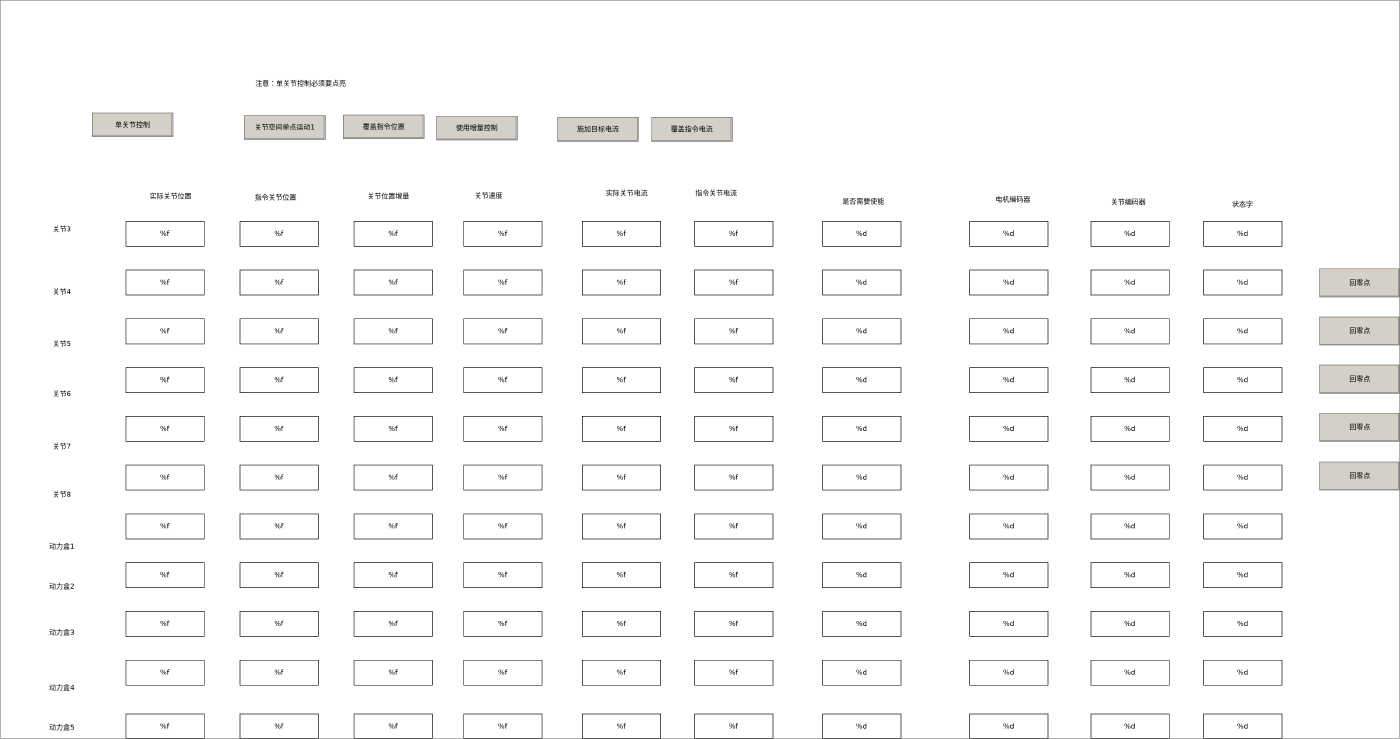
VISUALIZATION motion_a2  // 2208x1167
    Button (385,182 128x38), "关节空间单点运动1", colour toggle: g_motionTest.m_uiArmMode[2,1]
        tap g_motionTest.m_uiArmMode[1,1]
    Label (362,298 145x28), "指令关节位置"
    Label (194,295 150x30), "实际关节位置"
    Label (540,296 145x28), "关节位置增量"
    Label (698,295 145x28), "关节速度"
    Label (916,291 145x28), "实际关节电流"
    Label (1057,291 145x28), "指令关节电流"
    Rectangle (198,580 124x40), "%f", text variable: g_motionTest.m_actJntPos[2][1]
    Label (25,348 145x28), "关节3"
    Label (25,447 145x28), "关节4"
    Label (25,529 145x28), "关节5"
    Label (25,608 145x28), "关节6"
    Label (25,691 145x28), "关节7"
    Label (25,767 145x28), "关节8"
    Label (25,849 145x28), "动力盒1"
    Label (25,912 145x28), "动力盒2"
    Label (25,1135 145x28), "动力盒5"
    Label (25,985 145x28), "动力盒3"
    Label (25,1072 145x28), "动力盒4"
    Rectangle (198,657 124x40), "%f", text variable: g_motionTest.m_actJntPos[2][2]
    Rectangle (198,734 124x40), "%f", text variable: g_motionTest.m_actJntPos[2][3]
    Rectangle (198,811 124x40), "%f", text variable: g_motionTest.m_actJntPos[2][4]
    Rectangle (198,888 124x40), "%f", text variable: g_motionTest.m_actJntPos[2][5]
    Rectangle (198,965 124x40), "%f", text variable: g_motionTest.m_actJntPos[2][6]
    Rectangle (198,1042 124x40), "%f", text variable: g_motionTest.m_actJntPos[2][7]
    Rectangle (198,1127 124x40), "%f", text variable: g_motionTest.m_actJntPos[2][8]
    Rectangle (198,349 124x40), "%f", text variable: g_motionTest.m_actJntPosSetup[2][3]
    Rectangle (198,426 124x40), "%f", text variable: g_motionTest.m_actJntPosSetup[2][4]
    Rectangle (198,503 124x40), "%f", text variable: g_motionTest.m_actJntPosSetup[2][5]
    Rectangle (378,349 124x40), "%f", text variable: g_motionTest.m_targetJntPosSetup[2][3]
        OnMouseClick: write the text variable via Default
    Rectangle (378,426 124x40), "%f", text variable: g_motionTest.m_targetJntPosSetup[2][4]
        OnMouseClick: write the text variable via Default
    Rectangle (378,503 124x40), "%f", text variable: g_motionTest.m_targetJntPosSetup[2][5]
        OnMouseClick: write the text variable via Default
    Rectangle (378,580 124x40), "%f", text variable: g_motionTest.m_targetJntPosN8[2][1]
        OnMouseClick: write the text variable via Default
    Rectangle (378,657 124x40), "%f", text variable: g_motionTest.m_targetJntPosN8[2][2]
        OnMouseClick: write the text variable via Default
    Rectangle (378,734 124x40), "%f", text variable: g_motionTest.m_targetJntPosN8[2][3]
        OnMouseClick: write the text variable via Default
    Rectangle (378,811 124x40), "%f", text variable: g_motionTest.m_targetJntPosN8[2][4]
        OnMouseClick: write the text variable via Default
    Rectangle (378,888 124x40), "%f", text variable: g_motionTest.m_targetJntPosN8[2][5]
        OnMouseClick: write the text variable via Default
    Rectangle (378,965 124x40), "%f", text variable: g_motionTest.m_targetJntPosN8[2][6]
        OnMouseClick: write the text variable via Default
    Rectangle (378,1042 124x40), "%f", text variable: g_motionTest.m_targetJntPosN8[2][7]
        OnMouseClick: write the text variable via Default
    Rectangle (378,1127 124x40), "%f", text variable: g_motionTest.m_targetJntPosN8[2][8]
        OnMouseClick: write the text variable via Default
    Rectangle (558,349 124x40), "%f", text variable: g_motionTest.m_targetJntPosIncSetup[2][3]
        OnMouseClick: write the text variable via Default
    Rectangle (558,426 124x40), "%f", text variable: g_motionTest.m_targetJntPosIncSetup[2][4]
        OnMouseClick: write the text variable via Default
    Rectangle (558,503 124x40), "%f", text variable: g_motionTest.m_targetJntPosIncSetup[2][5]
        OnMouseClick: write the text variable via Default
    Rectangle (558,580 124x40), "%f", text variable: g_motionTest.m_targetJntPosIncN8[2][1]
        OnMouseClick: write the text variable via Default
    Rectangle (558,657 124x40), "%f", text variable: g_motionTest.m_targetJntPosIncN8[2][2]
        OnMouseClick: write the text variable via Default
    Rectangle (558,734 124x40), "%f", text variable: g_motionTest.m_targetJntPosIncN8[2][3]
        OnMouseClick: write the text variable via Default
    Rectangle (558,811 124x40), "%f", text variable: g_motionTest.m_targetJntPosIncN8[2][4]
        OnMouseClick: write the text variable via Default
    Rectangle (558,888 124x40), "%f", text variable: g_motionTest.m_targetJntPosIncN8[2][5]
        OnMouseClick: write the text variable via Default
    Rectangle (558,965 124x40), "%f", text variable: g_motionTest.m_targetJntPosIncN8[2][6]
        OnMouseClick: write the text variable via Default
    Rectangle (558,1042 124x40), "%f", text variable: g_motionTest.m_targetJntPosIncN8[2][7]
        OnMouseClick: write the text variable via Default
    Rectangle (558,1127 124x40), "%f", text variable: g_motionTest.m_targetJntPosIncN8[2][8]
        OnMouseClick: write the text variable via Default
    Rectangle (731,349 124x40), "%f", text variable: g_motionTest.m_targetJntVelSetup[2][3]
        OnMouseClick: write the text variable via Default
    Rectangle (731,426 124x40), "%f", text variable: g_motionTest.m_targetJntVelSetup[2][4]
        OnMouseClick: write the text variable via Default
    Rectangle (731,503 124x40), "%f", text variable: g_motionTest.m_targetJntVelSetup[2][5]
        OnMouseClick: write the text variable via Default
    Rectangle (731,580 124x40), "%f", text variable: g_motionTest.m_targetJntVel[2][1]
        OnMouseClick: write the text variable via Default
    Rectangle (731,657 124x40), "%f", text variable: g_motionTest.m_targetJntVel[2][2]
        OnMouseClick: write the text variable via Default
    Rectangle (731,734 124x40), "%f", text variable: g_motionTest.m_targetJntVel[2][3]
        OnMouseClick: write the text variable via Default
    Rectangle (731,811 124x40), "%f", text variable: g_motionTest.m_targetJntVel[2][4]
        OnMouseClick: write the text variable via Default
    Rectangle (731,888 124x40), "%f", text variable: g_motionTest.m_targetJntVel[2][5]
        OnMouseClick: write the text variable via Default
    Rectangle (731,965 124x40), "%f", text variable: g_motionTest.m_targetJntVel[2][6]
        OnMouseClick: write the text variable via Default
    Rectangle (731,1042 124x40), "%f", text variable: g_motionTest.m_targetJntVel[2][7]
        OnMouseClick: write the text variable via Default
    Rectangle (731,1127 124x40), "%f", text variable: g_motionTest.m_targetJntVel[2][8]
        OnMouseClick: write the text variable via Default
    Rectangle (918,349 124x40), "%f", text variable: g_motionTest.m_actJntCurrentSetup[2][3]
    Rectangle (918,426 124x40), "%f", text variable: g_motionTest.m_actJntCurrentSetup[2][4]
    Rectangle (918,503 124x40), "%f", text variable: g_motionTest.m_actJntCurrentSetup[2][5]
    Rectangle (918,580 124x40), "%f", text variable: g_motionTest.m_actJntCurrent[2][1]
    Rectangle (918,657 124x40), "%f", text variable: g_motionTest.m_actJntCurrent[2][2]
    Rectangle (918,734 124x40), "%f", text variable: g_motionTest.m_actJntCurrent[2][3]
    Rectangle (918,811 124x40), "%f", text variable: g_motionTest.m_actJntCurrent[2][4]
    Rectangle (918,888 124x40), "%f", text variable: g_motionTest.m_actJntCurrent[2][5]
    Rectangle (918,965 124x40), "%f", text variable: g_motionTest.m_actJntCurrent[2][6]
    Rectangle (918,1042 124x40), "%f", text variable: g_motionTest.m_actJntCurrent[2][7]
    Rectangle (918,1127 124x40), "%f", text variable: g_motionTest.m_actJntCurrent[2][8]
    Rectangle (1095,349 124x40), "%f", text variable: g_motionTest.m_targetJntCurrentSetup[2][3]
        OnMouseClick: write the text variable via Default
    Rectangle (1095,426 124x40), "%f", text variable: g_motionTest.m_targetJntCurrentSetup[2][4]
        OnMouseClick: write the text variable via Default
    Rectangle (1095,503 124x40), "%f", text variable: g_motionTest.m_targetJntCurrentSetup[2][5]
        OnMouseClick: write the text variable via Default
    Rectangle (1095,580 124x40), "%f", text variable: g_motionTest.m_targetJntCurrentN8[2][1]
        OnMouseClick: write the text variable via Default
    Rectangle (1095,657 124x40), "%f", text variable: g_motionTest.m_targetJntCurrentN8[2][2]
        OnMouseClick: write the text variable via Default
    Rectangle (1095,734 124x40), "%f", text variable: g_motionTest.m_targetJntCurrentN8[2][3]
        OnMouseClick: write the text variable via Default
    Rectangle (1095,811 124x40), "%f", text variable: g_motionTest.m_targetJntCurrentN8[2][4]
        OnMouseClick: write the text variable via Default
    Rectangle (1095,888 124x40), "%f", text variable: g_motionTest.m_targetJntCurrentN8[2][5]
        OnMouseClick: write the text variable via Default
    Rectangle (1095,965 124x40), "%f", text variable: g_motionTest.m_targetJntCurrentN8[2][6]
        OnMouseClick: write the text variable via Default
    Rectangle (1095,1042 124x40), "%f", text variable: g_motionTest.m_targetJntCurrentN8[2][7]
        OnMouseClick: write the text variable via Default
    Rectangle (1095,1127 124x40), "%f", text variable: g_motionTest.m_targetJntCurrentN8[2][8]
        OnMouseClick: write the text variable via Default
    Button (688,183 128x38), "使用增量控制", colour toggle: g_motionTest.m_singleMotorIncControl[2]
        toggle g_motionTest.m_singleMotorIncControl[2]
    Button (879,185 128x38), "施加目标电流", colour toggle: g_motionTest.m_uiArmMode[2,9]
        toggle g_motionTest.m_uiArmMode[2,9]
    Button (145,178 128x38), "单关节控制", colour toggle: g_motionTest.m_singleMotorControl[2]
        toggle g_motionTest.m_singleMotorControl[2]
    Label (364,117 220x30), "注意：单关节控制必须要点亮"
    Label (1289,303 145x30), "是否需要使能"
    Rectangle (1297,349 124x40), "%d", text variable: g_motionTest.m_jntEnableSetup[2][3]
        OnMouseClick: write the text variable via Default
    Rectangle (1297,426 124x40), "%d", text variable: g_motionTest.m_jntEnableSetup[2][4]
        OnMouseClick: write the text variable via Default
    Rectangle (1297,503 124x40), "%d", text variable: g_motionTest.m_jntEnableSetup[2][5]
        OnMouseClick: write the text variable via Default
    Rectangle (1297,580 124x40), "%d", text variable: g_motionTest.m_jntEnable[2][1]
        OnMouseClick: write the text variable via Default
    Rectangle (1297,657 124x40), "%d", text variable: g_motionTest.m_jntEnable[2][2]
        OnMouseClick: write the text variable via Default
    Label (1525,301 145x28), "电机编码器"
    Label (1707,305 145x28), "关节编码器"
    Label (1887,309 145x28), "状态字"
    Rectangle (1529,349 124x40), "%d", text variable: g_systemInfo.m_setupJntInfo[2,3].m_motorInput.m_motorEncoder
    Rectangle (1529,426 124x40), "%d", text variable: g_systemInfo.m_setupJntInfo[2,4].m_motorInput.m_motorEncoder
    Rectangle (1529,503 124x40), "%d", text variable: g_systemInfo.m_setupJntInfo[2,5].m_motorInput.m_motorEncoder
    Rectangle (1529,580 124x40), "%d", text variable: g_systemInfo.m_slaveJntInfo[2,1].m_motorInput.m_motorEncoder
    Rectangle (1529,657 124x40), "%d", text variable: g_systemInfo.m_slaveJntInfo[2,2].m_motorInput.m_motorEncoder
    Rectangle (1720,349 124x40), "%d", text variable: g_systemInfo.m_setupJntInfo[2,3].m_motorInput.m_linkEncoder
    Rectangle (1720,426 124x40), "%d", text variable: g_systemInfo.m_setupJntInfo[2,4].m_motorInput.m_linkEncoder
    Rectangle (1720,503 124x40), "%d", text variable: g_systemInfo.m_setupJntInfo[2,5].m_motorInput.m_linkEncoder
    Rectangle (1720,580 124x40), "%d", text variable: g_systemInfo.m_slaveJntInfo[2,1].m_motorInput.m_linkEncoder
    Rectangle (1720,657 124x40), "%d", text variable: g_systemInfo.m_slaveJntInfo[2,2].m_motorInput.m_linkEncoder
    Rectangle (1898,349 124x40), "%d", text variable: g_systemInfo.m_setupJntInfo[2,3].m_motorInput.m_statusWord
    Rectangle (1898,426 124x40), "%d", text variable: g_systemInfo.m_setupJntInfo[2,4].m_motorInput.m_statusWord
    Rectangle (1898,503 124x40), "%d", text variable: g_systemInfo.m_setupJntInfo[2,5].m_motorInput.m_statusWord
    Rectangle (1898,580 124x40), "%d", text variable: g_systemInfo.m_slaveJntInfo[2,1].m_motorInput.m_statusWord
    Rectangle (1898,657 124x40), "%d", text variable: g_systemInfo.m_slaveJntInfo[2,2].m_motorInput.m_statusWord
    Rectangle (1529,734 124x40), "%d", text variable: g_systemInfo.m_slaveJntInfo[2,3].m_motorInput.m_motorEncoder
    Rectangle (1529,811 124x40), "%d", text variable: g_systemInfo.m_slaveJntInfo[2,4].m_motorInput.m_motorEncoder
    Rectangle (1529,888 124x40), "%d", text variable: g_systemInfo.m_slaveJntInfo[2,5].m_motorInput.m_motorEncoder
    Rectangle (1529,965 124x40), "%d", text variable: g_systemInfo.m_slaveJntInfo[2,6].m_motorInput.m_motorEncoder
    Rectangle (1529,1042 124x40), "%d", text variable: g_systemInfo.m_slaveJntInfo[2,7].m_motorInput.m_motorEncoder
    Rectangle (1529,1127 124x40), "%d", text variable: g_systemInfo.m_slaveJntInfo[2,8].m_motorInput.m_motorEncoder
    Rectangle (1720,734 124x40), "%d", text variable: g_systemInfo.m_slaveJntInfo[2,3].m_motorInput.m_linkEncoder
    Rectangle (1720,811 124x40), "%d", text variable: g_systemInfo.m_slaveJntInfo[2,4].m_motorInput.m_linkEncoder
    Rectangle (1720,888 124x40), "%d", text variable: g_systemInfo.m_slaveJntInfo[2,5].m_motorInput.m_linkEncoder
    Rectangle (1720,965 124x40), "%d", text variable: g_systemInfo.m_slaveJntInfo[2,6].m_motorInput.m_linkEncoder
    Rectangle (1720,1042 124x40), "%d", text variable: g_systemInfo.m_slaveJntInfo[2,7].m_motorInput.m_linkEncoder
    Rectangle (1720,1127 124x40), "%d", text variable: g_systemInfo.m_slaveJntInfo[2,8].m_motorInput.m_linkEncoder
    Rectangle (1898,734 124x40), "%d", text variable: g_systemInfo.m_slaveJntInfo[2,3].m_motorInput.m_statusWord
    Rectangle (1898,811 124x40), "%d", text variable: g_systemInfo.m_slaveJntInfo[2,4].m_motorInput.m_statusWord
    Rectangle (1898,888 124x40), "%d", text variable: g_systemInfo.m_slaveJntInfo[2,5].m_motorInput.m_statusWord
    Rectangle (1898,965 124x40), "%d", text variable: g_systemInfo.m_slaveJntInfo[2,6].m_motorInput.m_statusWord
    Rectangle (1898,1042 124x40), "%d", text variable: g_systemInfo.m_slaveJntInfo[2,7].m_motorInput.m_statusWord
    Rectangle (1898,1127 124x40), "%d", text variable: g_systemInfo.m_slaveJntInfo[2,8].m_motorInput.m_statusWord
    Rectangle (1297,734 124x40), "%d", text variable: g_motionTest.m_jntEnable[2][3]
        OnMouseClick: write the text variable via Default
    Rectangle (1297,811 124x40), "%d", text variable: g_motionTest.m_jntEnable[2][4]
        OnMouseClick: write the text variable via Default
    Rectangle (1297,888 124x40), "%d", text variable: g_motionTest.m_jntEnable[2][5]
        OnMouseClick: write the text variable via Default
    Rectangle (1297,965 124x40), "%d", text variable: g_motionTest.m_jntEnable[2][6]
        OnMouseClick: write the text variable via Default
    Rectangle (1297,1042 124x40), "%d", text variable: g_motionTest.m_jntEnable[2][7]
        OnMouseClick: write the text variable via Default
    Rectangle (1297,1127 124x40), "%d", text variable: g_motionTest.m_jntEnable[2][8]
        OnMouseClick: write the text variable via Default
    Button (541,181 128x38), "覆盖指令位置", colour toggle: g_motionTest.m_coverCmdPos[2]
        tap g_motionTest.m_coverCmdPos[2]
    Button (2081,424 127x45), "回零点", colour toggle: g_motionTest.m_goHomeSetup[2][4]
        tap g_motionTest.m_goHomeSetup[2][4]
    Button (2081,500 127x45), "回零点", colour toggle: g_motionTest.m_goHomeSetup[2][5]
        tap g_motionTest.m_goHomeSetup[2][5]
    Button (2081,576 127x45), "回零点", colour toggle: g_motionTest.m_goHome[2][1]
        tap g_motionTest.m_goHome[2][1]
    Button (2081,652 127x45), "回零点", colour toggle: g_motionTest.m_goHome[2][2]
        tap g_motionTest.m_goHome[2][2]
    Button (2081,729 127x45), "回零点", colour toggle: g_motionTest.m_goHome[2][3]
        tap g_motionTest.m_goHome[2][3]
    Button (1027,185 128x38), "覆盖指令电流", colour toggle: g_motionTest.m_coverCmdCurrent[2]
        tap g_motionTest.m_coverCmdCurrent[2]
END_VISUALIZATION

(* stored: Version 1.1.0.1, ProductVersion 3.1.4024.11
   Visu motion_a2: Id {237bca9d-52b3-48ca-868c-f7fa47ef0763} *)
